PROGRAM Grabber_OOR
VAR
END_VAR

IF Shuttle.ExtensionComplete THEN
	
	IF Otto.PickupLocation1 AND (Shuttle.GrabberLoadNotInSight[1] OR Shuttle.GrabberLoadNotInGrabRange[1]) THEN
		
		Shuttle.Grabber_OOR		:= TRUE;
		
	ELSIF Otto.PickupLocation2 AND (Shuttle.GrabberLoadNotInSight[2] OR Shuttle.GrabberLoadNotInGrabRange[2]) THEN 
		
		Shuttle.Grabber_OOR		:= TRUE;
		
	ELSIF Otto.PickupLocation3 AND 
			(Shuttle.GrabberLoadNotInSight[1] OR Shuttle.GrabberLoadNotInSight[2]) THEN 	
				
		Shuttle.Grabber_OOR		:= TRUE;
		
	ELSE
		
		Shuttle.Grabber_OOR		:= FALSE;
	
	END_IF

ELSE
	
	Shuttle.Grabber_OOR		:= FALSE;

END_IF

END_PROGRAM

(* stored: Version 1.1.0.1, ProductVersion 3.1.4024.9
   POU Grabber_OOR: Id {e17853d1-322c-42bd-984c-bc69f6220ced}, SpecialFunc None *)
